# EPICS autosave request: sriApp/Db/sri_settings.req
$(P)UA
$(P)KVP
$(P)WATCHDOG_LENGTH
$(P)STANDBY
$(P)TIMER
$(P)AUTOKILL_LENGTH
